ABB RobotStudio station: Ex1_ver2.rspag

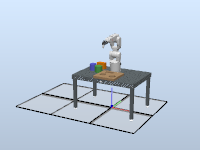
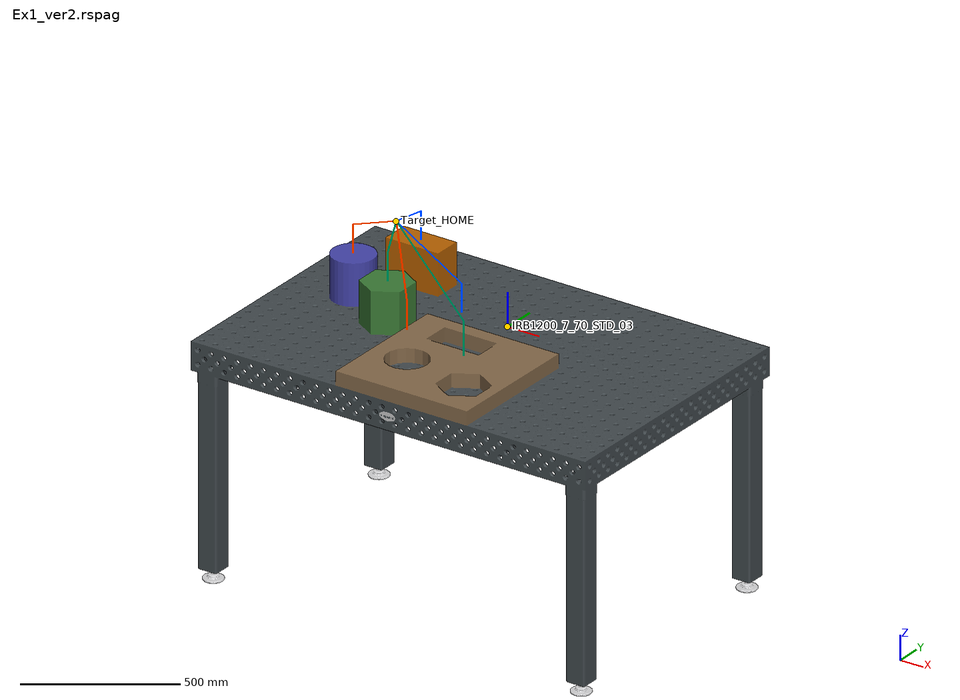
[picture v1: parts stored in the station drawn from their meshes, with robot base, taught points and paths (robot models come from the ABB library and are not in the file)]
--- station ---
Station Solution_1_Tutorial (saved by RobotStudio 21.4.9700.0)
Controller Controller1, task T_ROB1: task frame (RAPID world) sits at (0, 150, 830) mm, rotated rx 0 ry 0 rz -90 deg in the station
Controller Controller1
  mechanical unit ROB_1: IRB1200_7_70_STD_03, 6 joints, base frame (0, 0, 0) mm
Layout (positions relative to the parent item):
  - table [part] at (-200, -500, 830) mm, size 500 x 500 x 50 mm
  - object_1 [part] at (-600, -150, 830) mm, size 200 x 100 x 150 mm
  - object_2 [part] at (-650, -150, 830) mm, size 149.5 x 149.7 x 150 mm
  - object_3 [part] at (-700, -200, 830) mm, size 155.5 x 179.5 x 150 mm
  - siegmund_1500_1000 [part], size 1500 x 1010.3 x 830 mm
  - object_11 [part] at (-200, -500, 830) mm, size 200 x 100 x 150 mm
  - object_22 [part] at (-200, -500, 830) mm, size 149.5 x 149.7 x 150 mm
  - object_33 [part] at (-200, -500, 830) mm, size 155.5 x 179.5 x 150 mm
  - IRB1200_7_70_STD_03 [mechanism, from Robots\IRB1200_7_70_STD_03.rslib] at (0, 150, 830) mm, rotated rx 0 ry 0 rz -90 deg; joint values [0, 0, 0, 0, 0.5236, 0] (rad or m)
  - MyTool [mechanism, from Training Objects\myTool.rslib] at (0, -272.01, 1580.1) mm, rotated rx 180 ry 60 rz 90 deg
  - Positioner_OBJ1 [smart component, from Components\Positioner.rslib]
      properties: Object=object_1; Position=[-0.6 -0.15 0.83]; Orientation=[0 0 0]; Reference=Global; ReferenceObject=(none)
  - Positioner_OBJ2 [smart component, from Components\Positioner.rslib]
      properties: Object=object_2; Position=[-0.65 -0.15 0.83]; Orientation=[0 0 0]; Reference=Global; ReferenceObject=(none)
  - Positioner_OBJ3 [smart component, from Components\Positioner.rslib]
      properties: Object=object_3; Position=[-0.7 -0.2 0.83]; Orientation=[0 0 0]; Reference=Global; ReferenceObject=(none)
  - Attacher_OBJ1 [smart component, from Components\Attacher.rslib]
      properties: Parent=MyTool; Flange=0; Child=object_1; Mount=false; Offset=[0 0 0]; Orientation=[0 0 0]
  - Detacher_OBJ1 [smart component, from Components\Detacher.rslib]
      properties: Child=object_1; KeepPosition=true
  - Attacher_OBJ2 [smart component, from Components\Attacher.rslib]
      properties: Parent=MyTool; Flange=0; Child=object_2; Mount=false; Offset=[0 0 0]; Orientation=[0 0 0]
  - Detacher_OBJ2 [smart component, from Components\Detacher.rslib]
      properties: Child=object_2; KeepPosition=true
  - Attacher_OBJ3 [smart component, from Components\Attacher.rslib]
      properties: Parent=MyTool; Flange=0; Child=object_3; Mount=false; Offset=[0 0 0]; Orientation=[0 0 0]
  - Detacher_OBJ3 [smart component, from Components\Detacher.rslib]
      properties: Child=object_3; KeepPosition=true
Attachment: MyTool is attached to IRB1200_7_70_STD_03 / Link6
Station signals: DI DI_OBJ_POS
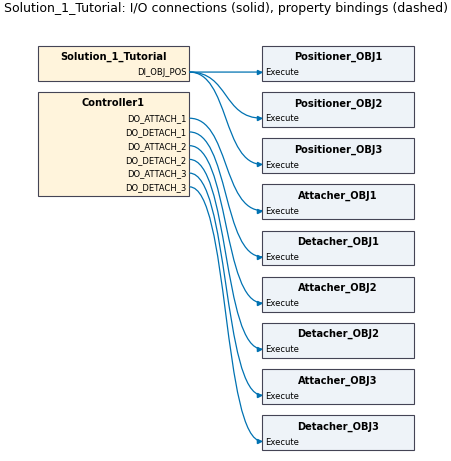
Station logic (signal -> signal, property => property):
  Solution_1_Tutorial.DI_OBJ_POS -> Positioner_OBJ1.Execute
  Solution_1_Tutorial.DI_OBJ_POS -> Positioner_OBJ2.Execute
  Solution_1_Tutorial.DI_OBJ_POS -> Positioner_OBJ3.Execute
  Controller1.DO_ATTACH_1 -> Attacher_OBJ1.Execute
  Controller1.DO_DETACH_1 -> Detacher_OBJ1.Execute
  Controller1.DO_ATTACH_2 -> Attacher_OBJ2.Execute
  Controller1.DO_DETACH_2 -> Detacher_OBJ2.Execute
  Controller1.DO_ATTACH_3 -> Attacher_OBJ3.Execute
  Controller1.DO_DETACH_3 -> Detacher_OBJ3.Execute

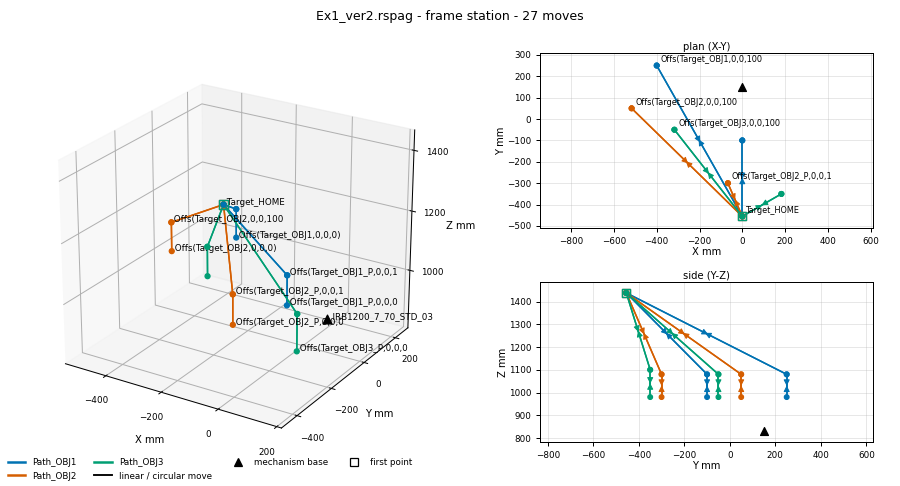
[picture p0: tool path of Ex1_ver2.rspag in frame station, 27 of 27 moves have a stored position in this frame; points joined in program order, loops and branches not executed]
--- Backups/Controller1/RAPID/TASK1/PROGMOD/CalibData.mod ---
MODULE CalibData
    PERS tooldata MyTool:=[TRUE,[[31.792631019,0,229.638935148],[0.945518576,0,0.325568154,0]],[1,[0,0,1],[1,0,0,0],0,0,0]];
ENDMODULE

--- Backups/Controller1/RAPID/TASK1/PROGMOD/Module1.mod ---
MODULE Module1
        CONST robtarget Target_HOME:=[[604.990919137,0,607.74730631],[0.190808996,0,0.981627183,0],[-1,0,-1,0],[9E+09,9E+09,9E+09,9E+09,9E+09,9E+09]];
    CONST robtarget Target_OBJ1:=[[-100,-400,150],[0,0.707106781,0.707106781,0],[-2,1,-2,0],[9E+09,9E+09,9E+09,9E+09,9E+09,9E+09]];
    CONST robtarget Target_OBJ1_P:=[[250,0,150],[0,0.707106781,0.707106781,0],[0,-1,1,0],[9E+09,9E+09,9E+09,9E+09,9E+09,9E+09]];
    CONST robtarget Target_OBJ2:=[[100,-517.298,150],[0,0.707106781,0.707106781,0],[-1,-2,1,0],[9E+09,9E+09,9E+09,9E+09,9E+09,9E+09]];
    CONST robtarget Target_OBJ2_P:=[[450,-67.298,150],[0,0.707106781,0.707106781,0],[0,-1,1,0],[9E+09,9E+09,9E+09,9E+09,9E+09,9E+09]];
    CONST robtarget Target_OBJ3:=[[200,-317.298,150],[0,0.707106781,0.707106781,0],[-1,-2,1,0],[9E+09,9E+09,9E+09,9E+09,9E+09,9E+09]];
    CONST robtarget Target_OBJ3_P:=[[500,182.702,150],[0,0.707106781,0.707106781,0],[0,-1,1,0],[9E+09,9E+09,9E+09,9E+09,9E+09,9E+09]];
!***********************************************************
    ! Description: Exercise 1 - complete vr.2 (with different robot and gripper)
    !
    ! Author: Karolina Kovarova
    !
!***********************************************************
     PROC main()
        Path_OBJ3;
        Path_OBJ2;
        Path_OBJ1;
    ENDPROC

    PROC Path_OBJ1()
        MoveL Target_HOME,v200,fine,MyTool\WObj:=wobj0;

        MoveL Offs(Target_OBJ1, 0, 0, 100),v200,fine,MyTool\WObj:=wobj0;
        MoveL Offs(Target_OBJ1, 0, 0, 0),v200,fine,MyTool\WObj:=wobj0;
        waitTime 0.1;
        PulseDO DO_ATTACH_1;
        waitTime 0.1;
        MoveL Offs(Target_OBJ1, 0, 0, 100),v200,fine,MyTool\WObj:=wobj0;

        MoveL Target_HOME,v200,fine,MyTool\WObj:=wobj0;

        MoveL Offs(Target_OBJ1_P, 0, 0, 100),v200,fine,MyTool\WObj:=wobj0;
        MoveL Offs(Target_OBJ1_P, 0, 0, 0),v200,fine,MyTool\WObj:=wobj0;
        waitTime 0.1;
        PulseDO DO_DETACH_1;
        waitTime 0.1;
        MoveL Offs(Target_OBJ1_P, 0, 0, 100),v200,fine,MyTool\WObj:=wobj0;

        MoveL Target_HOME,v200,fine,MyTool\WObj:=wobj0;
    ENDPROC

    PROC Path_OBJ2()
        MoveL Target_HOME,v200,fine,MyTool\WObj:=wobj0;

        MoveL Offs(Target_OBJ2, 0, 0, 100),v200,fine,MyTool\WObj:=wobj0;
        MoveL Offs(Target_OBJ2, 0, 0, 0),v200,fine,MyTool\WObj:=wobj0;
        waitTime 0.1;
        PulseDO DO_ATTACH_2;
        waitTime 0.1;
        MoveL Offs(Target_OBJ2, 0, 0, 100),v200,fine,MyTool\WObj:=wobj0;

        MoveL Target_HOME,v200,fine,MyTool\WObj:=wobj0;

        MoveL Offs(Target_OBJ2_P, 0, 0, 100),v200,fine,MyTool\WObj:=wobj0;
        MoveL Offs(Target_OBJ2_P, 0, 0, 0),v200,fine,MyTool\WObj:=wobj0;
        waitTime 0.1;
        PulseDO DO_DETACH_2;
        waitTime 0.1;
        MoveL Offs(Target_OBJ2_P, 0, 0, 100),v200,fine,MyTool\WObj:=wobj0;

        MoveL Target_HOME,v200,fine,MyTool\WObj:=wobj0;
    ENDPROC

    PROC Path_OBJ3()
        MoveL Target_HOME,v200,fine,MyTool\WObj:=wobj0;

        MoveL Offs(Target_OBJ3, 0, 0, 100),v200,fine,MyTool\WObj:=wobj0;
        MoveL Offs(Target_OBJ3, 0, 0, 0),v200,fine,MyTool\WObj:=wobj0;
        waitTime 0.1;
        PulseDO DO_ATTACH_3;
        waitTime 0.1;
        MoveL Offs(Target_OBJ3, 0, 0, 100),v200,fine,MyTool\WObj:=wobj0;

        MoveL Target_HOME,v200,fine,MyTool\WObj:=wobj0;

        MoveL Offs(Target_OBJ3_P, 0, 0, 120),v200,fine,MyTool\WObj:=wobj0;
        MoveL Offs(Target_OBJ3_P, 0, 0, 0),v200,fine,MyTool\WObj:=wobj0;
        waitTime 0.1;
        PulseDO DO_DETACH_3;
        waitTime 0.1;
        MoveL Offs(Target_OBJ3_P, 0, 0, 120),v200,fine,MyTool\WObj:=wobj0;

        MoveL Target_HOME,v200,fine,MyTool\WObj:=wobj0;
    ENDPROC
ENDMODULE

--- Backups/Controller1/SYSPAR/EIO.cfg ---
EIO:CFG_1.0:6:1::
#
EIO_SIGNAL:

      -Name "DO_ATTACH_1" -SignalType "DO"

      -Name "DO_ATTACH_2" -SignalType "DO"

      -Name "DO_ATTACH_3" -SignalType "DO"

      -Name "DO_DETACH_1" -SignalType "DO"

      -Name "DO_DETACH_2" -SignalType "DO"

      -Name "DO_DETACH_3" -SignalType "DO"
